FUNCTION_BLOCK FB_Motor_PT
VAR_INPUT
END_VAR
VAR_OUTPUT
END_VAR
VAR
	TempSensor					: I_TempSensor;
	nTemperature 				: REAL;
END_VAR

nTemperature := TempSensor.P_DegreesC;

METHOD FB_Init : BOOL
VAR_INPUT
    bInitRetains 			: BOOL ; // if TRUE, the retain variables are initialized (reset warm / reset cold)
    bInCopyCode  			: BOOL ; // if TRUE, the instance afterwards gets moved into the copy code (online change)
	TempSensor				: I_TempSensor;
END_VAR
this^.TempSensor := TempSensor;
END_METHOD

END_FUNCTION_BLOCK

(* stored: Version 1.1.0.1, ProductVersion 3.1.4024.12
   POU FB_Motor_PT: Id {6caff27d-6c1b-44a6-a830-e43bb9eb0ae4}, SpecialFunc None
   Method FB_Init: Id {2aa0dc3d-6dbf-49a8-be50-28e892b9218f} *)
